TYPE ST_Controller_Status :
STRUCT
	HasFault : BOOL;
	bEnabled : BOOL;
	Sensors : INT;
END_STRUCT
END_TYPE

(* stored: Version 1.1.0.1, ProductVersion 3.1.4024.16
   DUT ST_Controller_Status: Id {9a0878d7-f546-461b-9b25-bc057e9cf7ec} *)
